FUNCTION_BLOCK FB_XP_ProductData EXTENDS FB_CH_Object IMPLEMENTS I_XP_ProductData
VAR
	{attribute 'hide'}
	ipMover : I_XP_Mover_PLC;
END_VAR

{attribute 'monitoring':='call'}
PROPERTY LinkedMover : I_XP_Mover_PLC
GET
LinkedMover := ipMover;
END_GET
END_PROPERTY

METHOD LinkToMover : BOOL //it is not necessary to call this method. This is already done internally
VAR_INPUT
	ipMoverPlc : I_XP_Mover_PLC;
END_VAR
THIS^.ipMover := ipMoverPlc;
END_METHOD

END_FUNCTION_BLOCK

(* stored: Version 1.1.0.1, ProductVersion 3.1.4024.12
   POU FB_XP_ProductData: Id {c3b6a424-9c9b-4039-995e-b504f71b0675}, SpecialFunc None
   Property LinkedMover: Id {b33a3378-74c2-474f-b83f-666ab94dc90c}
   Get Get: Id {169be84a-95d3-41ec-ab28-fc2e7ac6853b}
   Method LinkToMover: Id {c64513f4-4ee1-4669-af43-579f90031b30} *)
